FUNCTION_BLOCK C_BINARYREADER
VAR_INPUT
END_VAR
VAR_OUTPUT
END_VAR
VAR
	_BASESTREAM 	: I_STREAM;
END_VAR

PROPERTY BASE_STREAM : I_STREAM
GET
Base_Stream := _BASESTREAM;
END_GET
END_PROPERTY

METHOD CLOSE : DINT
VAR_INPUT
END_VAR
Close := _BASESTREAM.Close();
_BASESTREAM := 0;
RETURN;
END_METHOD

METHOD NEW : DINT
VAR_INPUT
	STREAM : I_STREAM;
END_VAR
IF STREAM = 0 THEN
	New := 1;
	RETURN;
ELSE
	IF STREAM.IsValid THEN
		_BASESTREAM := STREAM;
		_BASESTREAM.Seek( 0, E_STREAMSEEKTYPE.Origin);
		New := -1;
		RETURN;
	ELSE
		New := 1;
		RETURN;
	END_IF
END_IF
END_METHOD

METHOD READ_BOOL : DINT
VAR_INPUT
	out_data : POINTER TO BOOL;
END_VAR
IF _BASESTREAM = 0 THEN
	Read_Bool := 1;
	RETURN;
END_IF

Read_Bool := _BASESTREAM.Read(out_data , 1);
RETURN;
END_METHOD

METHOD READ_BYTES : DINT
VAR_INPUT
	out_data 	: POINTER TO BYTE;
	length		: UDINT;
END_VAR
IF _BASESTREAM = 0 THEN
	Read_Bytes := 1;
	RETURN;
END_IF

Read_Bytes := _BASESTREAM.Read(out_data, length);
RETURN;
END_METHOD

METHOD READ_DOUBLE : DINT
VAR_INPUT
	out_data : POINTER TO LREAL;
END_VAR
IF _BASESTREAM = 0 THEN
	Read_Double := 1;
	RETURN;
END_IF

Read_Double := _BASESTREAM.Read(out_data , 8);
RETURN;
END_METHOD

METHOD READ_FLOAT : DINT
VAR_INPUT
	out_data : POINTER TO REAL;
END_VAR
IF _BASESTREAM = 0 THEN
	Read_Float := 1;
	RETURN;
END_IF

Read_Float := _BASESTREAM.Read(out_data , 4);
RETURN;
END_METHOD

METHOD READ_INT16 : DINT
VAR_INPUT
	out_data : POINTER TO INT;
END_VAR
IF _BASESTREAM = 0 THEN
	Read_Int16 := 1;
	RETURN;
END_IF

Read_Int16 := _BASESTREAM.Read(out_data , 2);
RETURN;
END_METHOD

METHOD READ_INT32 : DINT
VAR_INPUT
	out_data : POINTER TO DINT;
END_VAR
IF _BASESTREAM = 0 THEN
	Read_Int32 := 1;
	RETURN;
END_IF

Read_Int32 := _BASESTREAM.Read(out_data , 4);
RETURN;
END_METHOD

METHOD READ_STRING : DINT
VAR_INPUT
	out_data 	: PVOID;
	length		: UDINT;
END_VAR
IF _BASESTREAM = 0 THEN
	Read_String := 1;
	RETURN;
END_IF

Read_String := _BASESTREAM.Read(out_data, length);
RETURN;
END_METHOD

METHOD READ_UINT16 : DINT
VAR_INPUT
	out_data : POINTER TO UINT;
END_VAR
IF _BASESTREAM = 0 THEN
	Read_UInt16 := 1;
	RETURN;
END_IF

Read_UInt16 := _BASESTREAM.Read(out_data , 4);
RETURN;
END_METHOD

METHOD READ_UINT32 : DINT
VAR_INPUT
	out_data : POINTER TO UDINT;
END_VAR
IF _BASESTREAM = 0 THEN
	Read_UInt32 := 1;
	RETURN;
END_IF

Read_UInt32 := _BASESTREAM.Read(out_data , 4);
RETURN;
END_METHOD

END_FUNCTION_BLOCK

(* stored: Version 1.1.0.1, ProductVersion 3.1.4022.3
   POU C_BINARYREADER: Id {26d50fc3-a7d7-4aac-90e3-beef0b45fd3c}, SpecialFunc None
   Property BASE_STREAM: Id {cae1e64a-624a-421c-9265-d5478890aa63}
   Get Get: Id {0bf80ca8-bdb9-4fb6-8779-8150704bb550}
   Method CLOSE: Id {c74bc442-0074-4363-b6c5-e4cba1c44986}
   Method NEW: Id {4fab25d8-83ce-4e9c-9cc9-0faf6df608eb}
   Method READ_BOOL: Id {a87d9f12-f851-4142-baee-e60f10117a1c}
   Method READ_BYTES: Id {0f808161-3081-4dd1-99ea-54e31e636a75}
   Method READ_DOUBLE: Id {0930d98a-49cb-49a8-8b9a-c72cde6e8c27}
   Method READ_FLOAT: Id {e07b3f87-841b-4e43-8f63-a152b8522c0c}
   Method READ_INT16: Id {d91f549d-f034-409b-9b66-ed3c2adf39bb}
   Method READ_INT32: Id {69f6ce91-cdbb-4494-a298-67b14f02d373}
   Method READ_STRING: Id {9d704eee-d7d1-438b-ba04-0a39350bcebd}
   Method READ_UINT16: Id {7dea6d1b-2be9-4933-890b-f7a24a7f5e97}
   Method READ_UINT32: Id {c84d6b67-723e-4a02-a75a-a7d3c8267bd4} *)
